(* PLC project Generated.project, CODESYS CODESYS V3.5 SP19 Patch 1 *)
(* stored: creationDateTime 2026-10-27T16:00:37.967713, modificationDateTime 2026-10-27T16:00:37.967713 *)

(* ======================================================================= 📊 ST_Diag_Device — Structure diagnostic d'un esclave ou bus ─────────────────────────────────────────────────────────────── 🎯 Rôle : Structure de donnees d'état, diagnostic et alarme d'un equipement réseau 📄 Doc métier : DOC/AF/AF_Partie-12_Fonction_Diagnostic_v1.4.md ======================================================================= *)
TYPE ST_Diag_Device : STRUCT
  Online : BOOL;  (* Esclave visible sur le bus *)
  Operational : BOOL;  (* Esclave en mode OP (opérationnel) *)
  Error : BOOL;  (* Signal de défaut actif pour cet esclave *)
  ErrorId : WORD;  (* Code défaut détaillé *)
  State : E_Diag_State;  (* Phase courante du cycle de diagnostic *)
  StateAtError : E_Diag_State;  (* Instantané de la phase lors de l'anomalie *)
END_STRUCT;
END_TYPE

(* ======================================================================= 🧩 ST_Fault — Brique socle défaut (2 vues : live + latchée) ─────────────────────────────────────────────────────────────── 🎯 Rôle : porter l'état défaut d'un composant, applicable dans TOUS les cas (acquittable ou non), sans brique warning séparée. • Vue LIVE (Error / ErrorId) : suit la cause, retombe seule à 0. • Vue LATCHÉE (Latched / LatchedId): mémorisée au défaut, reste jusqu'au front Reset. Le choix acquittable / non-acquittable se fait PAR CAUSE (ST_FaultCause.Latching), jamais par bloc. 🔒 Sécurité : interlock TOUJOURS sur la cause brute (Error / ErrorId), jamais sur l'acquittement. Reset TOUJOURS effectif, jamais conditionné (std §9). 🧬 Composition : brique de base réutilisable — sortie de FB, struct métier, GVL. Texte IHM NON stocké ici : dérivé côté IHM depuis LatchedId / ErrorId. 📄 Doc : DOC/STDS/CODE_QUALITY_STANDARDS.md §2quinquies / §9 ======================================================================= *)
TYPE ST_Fault : STRUCT
  Error : BOOL;  (* <-- [DIAG] vue LIVE : au moins une cause présente maintenant *)
  ErrorId : WORD;  (* <-- [DIAG] bitfield des causes présentes maintenant (0 si aucune) *)
  Latched : BOOL;  (* <-- [DIAG] vue LATCHÉE : défaut non acquitté, reste jusqu'au front Reset *)
  LatchedId : WORD;  (* <-- [DIAG] ErrorId figé à l'apparition du défaut, effacé au Reset *)
END_STRUCT;
END_TYPE

(* ======================================================================= 🧩 ST_FaultCause — Cause élémentaire alimentant ST_Fault (socle FB_FaultCore) ─────────────────────────────────────────────────────────────── 🎯 Rôle : une cause exprimée EN CLAIR (BOOL + libellé), sans bitfield ni masque. Le FB métier remplit une liste (ARRAY[0..15] OF ST_FaultCause) ; le socle FB_FaultCore en déduit ST_Fault (vue live + vue latchée). 🔒 Sécurité : interlock TOUJOURS sur Active (cause brute), jamais sur le latch. Latching = TRUE → la cause ARME la vue latchée (défaut à acquitter). Latching = FALSE → la cause n'alimente que la vue live (retombe seule). Fail-safe : une cause laissée à Latching=FALSE reste visible en live — pour la rendre acquittable, il faut le déclarer explicitement. 📄 Doc : DOC/STDS/CODE_QUALITY_STANDARDS.md §2quinquies / §9 ======================================================================= *)
TYPE ST_FaultCause : STRUCT
  Active : BOOL;  (* 1 = cause présente maintenant (interlock sur cette valeur) *)
  Latching : BOOL;  (* 1 = cause à acquitter (arme Latched) ; 0 = live seulement *)
  Texte : STRING;  (* libellé prêt IHM (non stocké dans ST_Fault, dérivé côté IHM) *)
END_STRUCT;
END_TYPE

(* ======================================================================= 🕹️ ST_fbJoystick_AxisCmd — Consigne d'axe normalisée (sortie FB_Joystick) ─────────────────────────────────────────────────────────────── 🎯 Rôle : Structure de consigne d'axe produite par FB_Joystick. 📤 Champs : Enable, StartStop, SpeedTgt (%) + StepTgt (palier 1..5) + direction en bits (DirectionPositive/Negative, AtNeutral). SpeedTgt reste pour l'IHM, StepTgt pour la logique. 📄 Doc métier : DOC/AF/AF_Partie-08_Fonction_Joystick_v2.5.md ======================================================================= *)
TYPE ST_fbJoystick_AxisCmd : STRUCT
  Enable : BOOL;  (* === CONSIGNES DE PILOTAGE AXE === --> [CMD] Autorisation globale pipeline (FALSE=neutralisation, sorties coupees) *)
  StartStop : BOOL;  (* --> [CMD] Validation de mouvement (TRUE=acceleration, FALSE=deceleration/arret) *)
  SpeedTgt : REAL;  (* --> [CMD] Vitesse cible non signee (0...100 %, signe/sens donné par Direction) - IHM *)
  StepTgt : INT;  (* --> [CMD] Palier de vitesse (1..5, 0=arret) - logique/limitations (derive de SpeedTgt) *)
  DirectionNegative : BOOL;  (* --> [CMD] Direction joystick ou intension de gestuelle *)
  DirectionPositive : BOOL;  (* --> [CMD] Direction joystick ou intension de gestuelle *)
  AtNeutral : BOOL;  (* --> [CMD] TRUE si axes en zone morte (position centrale) *)
  Direction : INT;  (* === MONITORING IHM (derive des bits ci-dessus, jamais lu en interlock) === <-- [STAT] Sens -1=Rev / 0=Neutre / +1=Fwd (anim IHM fleche ; lu aussi logique treuils PRG_04) *)
  Deflection : INT;  (* <-- [STAT] Deflexion signee -100..+100 % (anim IHM jauge/barre) *)
END_STRUCT;
END_TYPE

(* ======================================================================= ⚙️ ST_fbJoystick_Cfg — Réglages regroupés de FB_Joystick ─────────────────────────────────────────────────────────────── 🎯 Rôle : porter en un bloc les 5 paramètres de conditionnement du geste (zone morte, temporisations homme-mort, marge défaut capteur). Passé à FB_Joystick via l'entrée `Cfg` — échange bloc IHM / persistant. 🧬 Pattern cfg : aligné sur ST_CycleCfg / ST_WinchCfg (préfixe ST_<Domaine>Cfg, instance persistante dans GVL_PERSISTENT, pont FB_CfgPersistBridge_* à venir). 📄 Doc métier : DOC/AF/AF_Partie-08_Fonction_Joystick_v2.5.md (§5bis) ======================================================================= *)
TYPE ST_fbJoystick_Cfg : STRUCT
  DeadbandRaw : INT := 300;  (* Zone morte en points ADC bruts (0..10000) *)
  NeutralHoldTime : TIME := TIME#100MS;  (* Maintien continu au neutre avant désarmement homme-mort *)
  DeadmanArmHoldTime : TIME := TIME#100MS;  (* Appui continu bouton requis pour armer le geste *)
  DeadmanArmGraceTime : TIME := TIME#3S;  (* Délai de grâce post-armement avant désarmement neutre *)
  RawOutOfRangeMargin : INT := 500;  (* Marge ADC autour des bornes [0..10000] avant défaut capteur (AF08 §5bis) *)
  SpeedStepTable : ST_SpeedStepTable;  (* Les initialiseurs imbriqués de STRUCT (notamment les ARRAY) ne sont pas acceptés par STruCpp/CODESYS dans une déclaration de type. La table est fournie par la configuration persistante de l'appelant. 🪜 Table seuils % -> palier (conversion au joystick, logique FB_Winch §5) *)
  SpeedStepHystMargin : REAL := 2;  (* Marge d'hystérésis palier (%) autour des seuils (anti-oscillation) *)
  Initialized : BOOL := FALSE;  (* 🚦 Flag restauration boot (interne pont FB_CfgPersistBridge_fbJoystick_Cfg) *)
END_STRUCT;
END_TYPE

(* values of E_Diag_State: DISABLED: Désactivé (surveillance non active); READY: Opérationnel réel, pas de défaut; INIT: Initialisation / Recherche de réseau; MONITORING: Surveillance active (états transitoires); ERROR: Anomalie de communication; SIMULATED: Bypass simulation ou bypass réseau IHM — pas le bus réel *)

{attribute 'qualified_only'}
{attribute 'strict'}
TYPE E_Diag_State : (DISABLED := 0, READY := 1, INIT := 2, MONITORING := 3, ERROR := 4, SIMULATED := 5);
END_TYPE

(* ======================================================================= 🪜 ST_SpeedStepTable — Table des paliers de vitesse contacteurs ─────────────────────────────────────────────────────────────── 🎯 Rôle : Structure de configuration des contacteurs et seuils par palier 📄 Doc métier : DOC/AF/AF_Partie-10_Fonction_Winch_v2.1.md ======================================================================= *)
TYPE ST_SpeedStepTable : STRUCT
  P1R1 : BOOL;  (* === PALIER 1 (VITESSE MINIMALE) === Contacteur 1 pour Palier 1 *)
  P1R2 : BOOL;  (* Contacteur 2 pour Palier 1 *)
  P1R3 : BOOL;  (* Contacteur 3 pour Palier 1 *)
  P1R4 : BOOL;  (* Contacteur 4 pour Palier 1 *)
  P2R1 : BOOL;  (* === PALIER 2 === Contacteur 1 pour Palier 2 *)
  P2R2 : BOOL;  (* Contacteur 2 pour Palier 2 *)
  P2R3 : BOOL;  (* Contacteur 3 pour Palier 2 *)
  P2R4 : BOOL;  (* Contacteur 4 pour Palier 2 *)
  P3R1 : BOOL;  (* === PALIER 3 === Contacteur 1 pour Palier 3 *)
  P3R2 : BOOL;  (* Contacteur 2 pour Palier 3 *)
  P3R3 : BOOL;  (* Contacteur 3 pour Palier 3 *)
  P3R4 : BOOL;  (* Contacteur 4 pour Palier 3 *)
  P4R1 : BOOL;  (* === PALIER 4 === Contacteur 1 pour Palier 4 *)
  P4R2 : BOOL;  (* Contacteur 2 pour Palier 4 *)
  P4R3 : BOOL;  (* Contacteur 3 pour Palier 4 *)
  P4R4 : BOOL;  (* Contacteur 4 pour Palier 4 *)
  P5R1 : BOOL;  (* === PALIER 5 (VITESSE MAXIMALE) === Contacteur 1 pour Palier 5 *)
  P5R2 : BOOL;  (* Contacteur 2 pour Palier 5 *)
  P5R3 : BOOL;  (* Contacteur 3 pour Palier 5 *)
  P5R4 : BOOL;  (* Contacteur 4 pour Palier 5 *)
  StepThreshold_Pct : ARRAY[1..5] OF REAL;  (* === SEUILS DE TRANSITION (%) === Seuils de changement de palier (0..100%) *)
END_STRUCT;
END_TYPE

(* ======================================================================= 🕹️ FB_Joystick — Acquisition & conditionnement du geste opérateur ─────────────────────────────────────────────────────────────── 🎯 Rôle : Acquisition 2 axes Hall + bouton homme-mort normatif. Pipeline par axe : FB_AxisScale -> Homme-Mort -> ST_fbJoystick_AxisCmd. 🔒 Sécurité : Armement homme-mort par maintien au neutre. Armement STRICTEMENT conditionné par ArmingPermit (permission externe, vue joystick) ; FALSE = armement bloqué + warning. Désarmement sur neutre prolongé ; le changement de mode / fin de cycle benne est géré par l'externe via ArmingPermit (vue joystick). 📤 Sorties : AxisCmdX/Y (struct = source unique : SpeedTgt NON signee % pour IHM + StepTgt palier 1..5 pour logique + bits sens + Direction -1/0/+1 et Deflection -100..+100 % pour anim IHM), Fault : ST_Fault (socle FB_FaultCore), AtNeutralXY (permis logique), NeutralXAct/YAct (miroirs IHM). 🧬 Contrat : `standard` — pas de struct métier propre → `Fault : ST_Fault` à plat. Pas de `State` (aucune machine d'état), pas de `ST_Lifecycle` (FB synchrone). ⚙️ Réglages regroupés dans `Cfg : ST_fbJoystick_Cfg` (échange bloc IHM / persistant). 📄 Doc métier : DOC/AF/AF_Partie-08_Fonction_Joystick_v2.5.md (F08.01, F08.03-F08.07) ===================================================================== *)
FUNCTION_BLOCK FB_Joystick
  VAR_INPUT
    Enable : BOOL;  (* === CONTRAT STANDARD (Enable + Reset) === --> [CMD] Active la logique du bloc (TRUE=Autorise) *)
    Reset : BOOL;  (* --> [CMD] Acquittement defaut (front, jamais conditionne) *)
    ArmingPermit : BOOL;  (* === PERMIS SECURITE === --> [SAFE] Permission d'armement homme-mort ; FALSE = armement bloqué *)
    DirectInversionPermit : BOOL;  (* --> [SAFE] Inversion Y sans neutre, semi-auto AX8..AX12 et repli du vidage AX15b *)
    BusCanOpenOP : ST_Diag_Device;  (* === ACQUISITION MATERIELLE & DIAGNOSTIC === --> [HW] Etat presence noeud CAN *)
    JoystickOP : ST_Diag_Device;  (* --> [HW] Mode esclave CANopen actif *)
    RawX : INT;  (* --> [HW] Valeur brute axe X (0..10000) *)
    RawY : INT;  (* --> [HW] Valeur brute axe Y (0..10000) *)
    RawButton : BOOL;  (* --> [HW] Etat brut bouton homme-mort *)
    Calibrate : BOOL;  (* === COMMANDES OPERATEUR & CALIBRATION === --> [CMD] Front : lance la calibration (recalage du neutre) *)
    Cfg : ST_fbJoystick_Cfg;  (* === REGLAGES & CONFIGURATION === --> [CFG] Réglages groupés (deadband, temporisations, marge ADC) *)
  END_VAR
  VAR_OUTPUT
    Ready : BOOL;  (* === CONTRAT STANDARD (Ready + Fault) === <-- [STAT] FB pret a fonctionner (Enable + bus OK + pas de defaut late) *)
    Fault : ST_Fault;  (* <-- [DIAG] Brique defaut socle (live + latche), remplie par FB_FaultCore *)
    AxisCmdX : ST_fbJoystick_AxisCmd;  (* === CONSIGNES AXES NORMALISEES === <-- [ACT] Consigne axe X : SpeedTgt (non signee 0..100) + bits sens + Direction/Deflection (monitoring) *)
    AxisCmdY : ST_fbJoystick_AxisCmd;  (* <-- [ACT] Consigne axe Y : SpeedTgt (non signee 0..100) + bits sens + Direction/Deflection (monitoring) *)
    DeadmanArmed : BOOL;  (* === HOMME-MORT === <-- [STAT] Geste arme (bouton maintenu + ArmingPermit) - IHM/diagnostic *)
    ArmingPermitDenied : BOOL;  (* <-- [DIAG] Appui homme-mort refuse (ArmingPermit=FALSE) - warning non latche (F08.08) *)
    AtNeutralXY : BOOL;  (* === ETAT LOGIQUE === <-- [STAT] Les 2 axes en zone morte BRUTE (ScaleX/Y.OutPct=0, AVANT homme-mort) - permis mouvement, LU EN LOGIQUE (PRG_03/04/07) *)
    NeutralXAct : INT;  (* === MIROIRS IHM / TEST === <-- [STAT] Point neutre X calibre courant *)
    NeutralYAct : INT;  (* <-- [STAT] Point neutre Y calibre courant *)
  END_VAR
  VAR_IN_OUT
    NeutralXMem : INT;  (* === RETENTION & CALIBRATION PERSISTANTE === <-> [BUS] Point neutre X persistant global *)
    NeutralYMem : INT;  (* <-> [BUS] Point neutre Y persistant global *)
  END_VAR
  VAR
    CST_DirectionQualificationThreshold_Pct : REAL := 0.1;  (* Seuil % : axe actif (StartStop / bits sens / palier 0) *)
    CST_InversionFlipThreshold_Pct : REAL := 10;  (* Seuil % : sens RETENU pour la détection d'inversion inter-scan. *)
    ScaleX : FB_AxisScale;  (* === SOUS-INSTANCES FB & TIMERS === * [INST] Normalisation et zone morte axe X *)
    ScaleY : FB_AxisScale;  (* * [INST] Normalisation et zone morte axe Y *)
    DeadmanEdge : R_TRIG;  (* * [INST] Detecteur front montant bouton homme-mort *)
    NeutralXYEdge : R_TRIG;  (* * [INST] Front retour simultane X+Y au neutre (libere verrou inversion) *)
    NeutralHoldTimer : TON;  (* * [INST] Temporisation maintien au neutre *)
    DeadmanArmTimer : TON;  (* * [INST] Temporisation maintien bouton armement *)
    DeadmanArmGraceTimer : TON;  (* * [INST] Temporisation delai de grace post-armement *)
    instFault : FB_FaultCore;  (* * [INST] Socle de defaut (liste de causes -> ST_Fault) *)
    SpeedStepHyst1 : HYSTERESIS;  (* * [INST] Decodage % -> palier, seuil 1 (logique FB_Winch §5) *)
    SpeedStepHyst2 : HYSTERESIS;  (* * [INST] Decodage % -> palier, seuil 2 *)
    SpeedStepHyst3 : HYSTERESIS;  (* * [INST] Decodage % -> palier, seuil 3 *)
    SpeedStepHyst4 : HYSTERESIS;  (* * [INST] Decodage % -> palier, seuil 4 *)
    CmdXVal : REAL;  (* === VARIABLES LOCALES INTERNES === . [LOC] Consigne axe X calculee apres filtrage/homme-mort *)
    CmdYVal : REAL;  (* . [LOC] Consigne axe Y calculee apres filtrage/homme-mort *)
    LastCalibrate : BOOL;  (* . [LOC] Memorisation etat precedent commande Calibrate (front) *)
    DeadmanArmPending : BOOL;  (* . [LOC] Armement en cours d'attente de la temporisation maintien *)
    InversionLockActive : BOOL;  (* . [LOC] Verrou retour neutre apres inversion inter-scan directe *)
    PrevDirX : INT;  (* . [LOC] Sens X qualifie au scan precedent (-1, 0, +1) *)
    PrevDirY : INT;  (* . [LOC] Sens Y qualifie au scan precedent (-1, 0, +1) *)
    DirX : INT;  (* . [LOC] Sens X qualifie au scan courant (-1, 0, +1) *)
    DirY : INT;  (* . [LOC] Sens Y qualifie au scan courant (-1, 0, +1) *)
    FlipX : BOOL;  (* . [LOC] Inversion X directe sans echantillon neutre *)
    FlipY : BOOL;  (* . [LOC] Inversion Y directe sans echantillon neutre *)
    RawOutOfRange : BOOL;  (* . [LOC] Surveillance capteur continue (AF08 §5bis) : RawX/RawY hors plage nominale+marge *)
    CalibFail : BOOL;  (* . [LOC] Echec calibration (front Calibrate hors zone) - cause a acquitter (latching) *)
    BusLost : BOOL;  (* . [LOC] Perte liaison bus / device non operationnel - cause live seulement *)
    instCauses : ARRAY[0..15] OF ST_FaultCause;  (* . [LOC] Liste des causes pour le socle FB_FaultCore *)
  END_VAR

            

{region "§1 CAUSES + SOCLE (appele AVANT le gate)"}
// 🎯 CAUSES exprimées en CLAIR (liste ST_FaultCause) — plus de bitfield WORD.
//    - CalibFail : cause A ACQUITTER (Latching=TRUE) -> arme Fault.Latched.
//    - RawOutOfRange / BusLost : cause LIVE seulement (Latching=FALSE) -> Fault.Error, retombe seule.
//    Interlock sur la cause brute ; le socle gère latch/reset.
RawOutOfRange := (RawX < (0 - Cfg.RawOutOfRangeMargin))
              OR (RawX > (10000 + Cfg.RawOutOfRangeMargin))
              OR (RawY < (0 - Cfg.RawOutOfRangeMargin))
              OR (RawY > (10000 + Cfg.RawOutOfRangeMargin));
BusLost := (NOT BusCanOpenOP.Operational OR NOT JoystickOP.Operational);

// Calibration : un front (Calibrate) hors zone -> cause a acquitter. La cause reste active tant que
// les axes sont HORS zone valide [2000..8000] : Reset ne l'efface que si la cause a disparu
// (interlock socle sur la cause brute). Effacee par un Reset avec axes en zone.
IF Calibrate AND NOT LastCalibrate THEN
    IF RawX >= 2000 AND RawX <= 8000 AND RawY >= 2000 AND RawY <= 8000 THEN
        NeutralXMem := RawX;       // memorisation nouvelle position neutre X
        NeutralYMem := RawY;       // memorisation nouvelle position neutre Y
        CalibFail := FALSE;        // calibration valide : plus de cause
    ELSE
        CalibFail := TRUE;         // échec : cause a acquitter (persistante tant que hors zone)
    END_IF;
END_IF;
LastCalibrate := Calibrate;
// Ré-acquisition de la cause (front Reset + cause disparue) : n'efface la cause QUE si les
// axes sont revenus en zone valide. Reste latee tant que hors zone (interlock sur cause brute).
IF Reset AND (RawX >= 2000 AND RawX <= 8000 AND RawY >= 2000 AND RawY <= 8000) THEN
    CalibFail := FALSE;
END_IF;

// Remplissage de la LISTE de causes pour le socle (index 0..2)
// Cause en clair (Active/Latching/Texte) ; 3 causes fixes.
instCauses[0].Active := CalibFail;     instCauses[0].Latching := TRUE;
instCauses[0].Texte := 'Echec calibration joystick (RawX/Y hors zone)';
instCauses[1].Active := RawOutOfRange; instCauses[1].Latching := FALSE;
instCauses[1].Texte := 'Capteur joystick hors plage ADC';
instCauses[2].Active := BusLost;       instCauses[2].Latching := FALSE;
instCauses[2].Texte := 'Perte liaison bus CAN joystick';

// Appel du socle TOUJOURS (meme si le gate RETURN ensuite) : la cause bus doit etre vue.
instFault(Enable := Enable, Reset := Reset, Causes := instCauses);
Fault := instFault.Fault;     // source de verite = socle

// Disponibilite = Enable + bus OK + pas de defaut LATE. Une cause live (bus, capteur) ne latche pas
// -> elle n'entre pas dans Fault.Latched ; le bus est deja couvert par ...OP.Operational ci-dessous.
Ready := Enable AND BusCanOpenOP.Operational AND JoystickOP.Operational AND NOT Fault.Latched;
{endregion}

{region "§2 Gate securite (neutralisation pipeline, n efface pas le statut)"}
// 1. GATE — neutralise le pipeline si indisponible. Le statut a deja ete rempli (zone 0).
IF NOT Enable OR BusLost THEN
    AxisCmdX.Enable := FALSE; AxisCmdX.StartStop := FALSE; AxisCmdX.SpeedTgt := 0.0; AxisCmdX.StepTgt := 0;
    AxisCmdX.DirectionPositive := FALSE; AxisCmdX.DirectionNegative := FALSE; AxisCmdX.AtNeutral := TRUE;
    AxisCmdY.Enable := FALSE; AxisCmdY.StartStop := FALSE; AxisCmdY.SpeedTgt := 0.0; AxisCmdY.StepTgt := 0;
    AxisCmdY.DirectionPositive := FALSE; AxisCmdY.DirectionNegative := FALSE; AxisCmdY.AtNeutral := TRUE;
    AxisCmdX.Direction := 0; AxisCmdX.Deflection := 0;
    AxisCmdY.Direction := 0; AxisCmdY.Deflection := 0;
    AtNeutralXY := TRUE;
    DeadmanArmed := FALSE;
    DeadmanArmPending := FALSE;
    InversionLockActive := FALSE;
    PrevDirX := 0;
    PrevDirY := 0;
    ArmingPermitDenied := FALSE;
    NeutralXYEdge(CLK := FALSE);
    NeutralHoldTimer(IN := FALSE, PT := Cfg.NeutralHoldTime);
    DeadmanArmTimer(IN := FALSE, PT := Cfg.DeadmanArmHoldTime);
    DeadmanArmGraceTimer(IN := FALSE, PT := Cfg.DeadmanArmGraceTime);
    NeutralXAct := NeutralXMem;
    NeutralYAct := NeutralYMem;
    RETURN;
END_IF;
{endregion}

{region "§3 Acquisition + mise a l echelle"}
// Mise a l'echelle (deadband) - le neutre s'evalue sur les 2 axes
ScaleX(RawIn := RawX, Neutral := NeutralXMem, DeadbandRaw := Cfg.DeadbandRaw);
ScaleY(RawIn := RawY, Neutral := NeutralYMem, DeadbandRaw := Cfg.DeadbandRaw);
AtNeutralXY := (ScaleX.OutPct = 0.0) AND (ScaleY.OutPct = 0.0);   // les 2 axes en zone morte - permis mouvement
{endregion}

{region "§4 Armement homme mort"}
// 🔀 Inversion inter-scan : le sens n'est RETENU que si la déflexion dépasse
// CST_InversionFlipThreshold_Pct (>> bruit Hall / bord de deadband). Un aller-retour
// +1<->-1 sans échantillon 0 pose le verrou. Levé exclusivement au front AtNeutralXY.
// RawOutOfRange : lecture capteur non fiable -> aucun sens retenu (le geste est déjà forcé à 0
// par le SEL du pipeline). Une reprise capteur-défaut -> valide ne compte donc pas comme flip.
DirX := 0;
DirY := 0;
IF NOT RawOutOfRange THEN
    IF ScaleX.OutPct > CST_InversionFlipThreshold_Pct THEN
        DirX := 1;
    ELSIF ScaleX.OutPct < -CST_InversionFlipThreshold_Pct THEN
        DirX := -1;
    END_IF;
    IF ScaleY.OutPct > CST_InversionFlipThreshold_Pct THEN
        DirY := 1;
    ELSIF ScaleY.OutPct < -CST_InversionFlipThreshold_Pct THEN
        DirY := -1;
    END_IF;
END_IF;
FlipX := ((PrevDirX = 1) AND (DirX = -1)) OR ((PrevDirX = -1) AND (DirX = 1));
FlipY := ((PrevDirY = 1) AND (DirY = -1)) OR ((PrevDirY = -1) AND (DirY = 1));

NeutralXYEdge(CLK := AtNeutralXY);
IF NeutralXYEdge.Q THEN
    InversionLockActive := FALSE;
END_IF;

IF FlipX OR (FlipY AND NOT (DirectInversionPermit AND DeadmanArmed)) THEN
    InversionLockActive := TRUE;
    DeadmanArmed := FALSE;
    DeadmanArmPending := FALSE;
END_IF;

// Bouton homme-mort : armement par MAINTIEN (Cfg.DeadmanArmHoldTime), independant de la position.
// ⚠️ Un appui PENDANT le verrou d'inversion n'arme PAS de demande : le nouveau front conscient
//    doit survenir APRÈS le retour au neutre (sinon on "pré-charge" le réarmement stick inversé).
DeadmanEdge(CLK := RawButton);
IF DeadmanEdge.Q AND NOT InversionLockActive THEN DeadmanArmPending := TRUE; END_IF;
IF NOT RawButton THEN DeadmanArmPending := FALSE; END_IF;

// Securite : armage UNIQUEMENT si DeadmanArmPending ET ArmingPermit.
DeadmanArmTimer(IN := DeadmanArmPending AND NOT DeadmanArmed AND ArmingPermit AND NOT InversionLockActive, PT := Cfg.DeadmanArmHoldTime);
IF DeadmanArmTimer.Q THEN
    DeadmanArmed := TRUE;
    DeadmanArmPending := FALSE;
END_IF;

// Désarmement externe immédiat : le retrait d'ArmingPermit (changement de mode, fin de cycle
// benne) désarme TOUT DE SUITE le geste — pas d'armement résiduel "surprise" à la ré-acquisition.
IF NOT ArmingPermit THEN
    DeadmanArmed := FALSE;
    DeadmanArmPending := FALSE;
END_IF;

// Avertissement "armage non autorise" (niveau, pendant l'appui non autorise)
ArmingPermitDenied := RawButton AND NOT ArmingPermit;

// Desarmage par maintien au neutre (apres grace)
DeadmanArmGraceTimer(IN := DeadmanArmed, PT := Cfg.DeadmanArmGraceTime);
NeutralHoldTimer(IN := DeadmanArmed AND AtNeutralXY AND DeadmanArmGraceTimer.Q, PT := Cfg.NeutralHoldTime);
IF NeutralHoldTimer.Q THEN DeadmanArmed := FALSE; END_IF;
{endregion}

{region "§5 Pipeline axe X"}
CmdXVal := SEL(DeadmanArmed AND NOT RawOutOfRange, 0.0, ScaleX.OutPct);

AxisCmdX.Enable := NOT RawOutOfRange AND ArmingPermit;
AxisCmdX.SpeedTgt := ABS(CmdXVal);   // NON signee (le sens = bits DirectionPositive/Negative + AxisCmdX.Direction)
AxisCmdX.StartStop := (ABS(CmdXVal) > CST_DirectionQualificationThreshold_Pct);

AxisCmdX.DirectionPositive := (CmdXVal > CST_DirectionQualificationThreshold_Pct);
AxisCmdX.DirectionNegative := (CmdXVal < -CST_DirectionQualificationThreshold_Pct);
AxisCmdX.AtNeutral := NOT AxisCmdX.DirectionPositive AND NOT AxisCmdX.DirectionNegative;
IF AxisCmdX.AtNeutral THEN AxisCmdX.SpeedTgt := 0.0; END_IF;

// Projections monitoring dans le struct (les bits restent la source logique)
IF AxisCmdX.DirectionPositive THEN AxisCmdX.Direction := 1;
ELSIF AxisCmdX.DirectionNegative THEN AxisCmdX.Direction := -1;
ELSE AxisCmdX.Direction := 0; END_IF;
AxisCmdX.Deflection := REAL_TO_INT(CmdXVal);   // deflexion signee -100..+100 % (anim IHM)
{endregion}

{region "§6 Pipeline axe Y et sorties"}
CmdYVal := SEL(DeadmanArmed AND NOT RawOutOfRange, 0.0, ScaleY.OutPct);

AxisCmdY.Enable := NOT RawOutOfRange AND ArmingPermit;
AxisCmdY.SpeedTgt := ABS(CmdYVal);   // NON signee (le sens = bits DirectionPositive/Negative + AxisCmdY.Direction)
AxisCmdY.StartStop := (ABS(CmdYVal) > CST_DirectionQualificationThreshold_Pct);

AxisCmdY.DirectionPositive := (CmdYVal > CST_DirectionQualificationThreshold_Pct);
AxisCmdY.DirectionNegative := (CmdYVal < -CST_DirectionQualificationThreshold_Pct);
AxisCmdY.AtNeutral := NOT AxisCmdY.DirectionPositive AND NOT AxisCmdY.DirectionNegative;
IF AxisCmdY.AtNeutral THEN AxisCmdY.SpeedTgt := 0.0; END_IF;

// 🪜 Decodage consigne % -> palier (logique FB_Winch §5, deplacee au joystick).
//    AxisCmdY.SpeedTgt (%) reste pour l'IHM ; AxisCmdY.StepTgt (1..5, 0=arret) pour la logique/limitations.
SpeedStepHyst1(IN := REAL_TO_INT(AxisCmdY.SpeedTgt), HIGH := REAL_TO_INT(Cfg.SpeedStepTable.StepThreshold_Pct[1] + Cfg.SpeedStepHystMargin), LOW := REAL_TO_INT(Cfg.SpeedStepTable.StepThreshold_Pct[1] - Cfg.SpeedStepHystMargin));
SpeedStepHyst2(IN := REAL_TO_INT(AxisCmdY.SpeedTgt), HIGH := REAL_TO_INT(Cfg.SpeedStepTable.StepThreshold_Pct[2] + Cfg.SpeedStepHystMargin), LOW := REAL_TO_INT(Cfg.SpeedStepTable.StepThreshold_Pct[2] - Cfg.SpeedStepHystMargin));
SpeedStepHyst3(IN := REAL_TO_INT(AxisCmdY.SpeedTgt), HIGH := REAL_TO_INT(Cfg.SpeedStepTable.StepThreshold_Pct[3] + Cfg.SpeedStepHystMargin), LOW := REAL_TO_INT(Cfg.SpeedStepTable.StepThreshold_Pct[3] - Cfg.SpeedStepHystMargin));
SpeedStepHyst4(IN := REAL_TO_INT(AxisCmdY.SpeedTgt), HIGH := REAL_TO_INT(Cfg.SpeedStepTable.StepThreshold_Pct[4] + Cfg.SpeedStepHystMargin), LOW := REAL_TO_INT(Cfg.SpeedStepTable.StepThreshold_Pct[4] - Cfg.SpeedStepHystMargin));

// ⚠️ HYSTERESIS (Util CODESYS) est un hystérésis BAS : OUT=TRUE quand IN<LOW, OUT=FALSE
//    quand IN>HIGH. Pour un décodage ASCENDANT (petite déflexion → palier bas, grande →
//    palier haut) on teste donc `NOT OUT` : palier supérieur seulement une fois IN au-dessus
//    du seuil (bande d'hystérésis LOW..HIGH autour de StepThreshold_Pct[n]).
IF AxisCmdY.SpeedTgt <= CST_DirectionQualificationThreshold_Pct THEN
    AxisCmdY.StepTgt := 0;
ELSE
    AxisCmdY.StepTgt := 1;
    IF NOT SpeedStepHyst1.OUT THEN AxisCmdY.StepTgt := 2; END_IF;
    IF NOT SpeedStepHyst2.OUT THEN AxisCmdY.StepTgt := 3; END_IF;
    IF NOT SpeedStepHyst3.OUT THEN AxisCmdY.StepTgt := 4; END_IF;
    IF NOT SpeedStepHyst4.OUT THEN AxisCmdY.StepTgt := 5; END_IF;
END_IF;

// Projections monitoring dans le struct (les bits restent la source logique)
IF AxisCmdY.DirectionPositive THEN AxisCmdY.Direction := 1;
ELSIF AxisCmdY.DirectionNegative THEN AxisCmdY.Direction := -1;
ELSE AxisCmdY.Direction := 0; END_IF;
AxisCmdY.Deflection := REAL_TO_INT(CmdYVal);   // deflexion signee -100..+100 % (anim IHM)

// Memorisation apres traitement : l'inversion suivante compare deux scans qualifies successifs.
PrevDirX := DirX;
PrevDirY := DirY;

// Miroirs point neutre courant
NeutralXAct := NeutralXMem;
NeutralYAct := NeutralYMem;
{endregion}

          
END_FUNCTION_BLOCK

(* ======================================================================= ⚙️ FB_AxisScale — Normalisation et zone morte d'un axe joystick ─────────────────────────────────────────────────────────────── 🎯 Rôle : Normalise une valeur brute (0..10000) selon le neutre calibré et applique une zone morte en unités brutes (compte ADC). 🛡️ Garde-fou : Saturation stricte de la consigne à +/-100.0 %. 📄 Doc métier : DOC/AF/AF_Partie-08_Fonction_Joystick_v2.5.md (F08.02) ======================================================================= *)
FUNCTION_BLOCK FB_AxisScale
  VAR_INPUT
    RawIn : INT;  (* === ENTRÉES MESURÉES & CONFIGURATION === --> [HW] Valeur brute potentiometre/Hall (0..10000) *)
    Neutral : INT;  (* --> [CFG] Point milieu calibre (compte brut ADC) *)
    DeadbandRaw : INT;  (* --> [CFG] Zone morte en unites brutes ADC (ex: 300) *)
  END_VAR
  VAR_OUTPUT
    OutPct : REAL;  (* === CONSIGNES CALCULÉES === <-- [STAT] Consigne d'axe mise a l'echelle (-100.0..+100.0 %) *)
  END_VAR
  VAR
    Delta : REAL;  (* === VARIABLES LOCALES INTERNES === . [LOC] Amplitude utile de la demi-plage d'axe *)
  END_VAR

            

IF RawIn >= Neutral THEN
    Delta := INT_TO_REAL(10000 - Neutral);
    IF Delta > 0.0 THEN
        OutPct := (INT_TO_REAL(RawIn - Neutral) / Delta) * 100.0;
    ELSE
        OutPct := 0.0;
    END_IF;
ELSE
    Delta := INT_TO_REAL(Neutral);
    IF Delta > 0.0 THEN
        OutPct := (INT_TO_REAL(RawIn - Neutral) / Delta) * 100.0;
    ELSE
        OutPct := 0.0;
    END_IF;
END_IF;

IF ABS(RawIn - Neutral) <= DeadbandRaw THEN
    OutPct := 0.0;
END_IF;

// 🛡️ Limitation de plage : une valeur brute hors plage nominale ne doit jamais
// produire une consigne supérieure à ±100 %. Ce garde-fou protège les
// consommateurs en aval, notamment la translation M3.
OutPct := LIMIT(-100.0, OutPct, 100.0);

          
END_FUNCTION_BLOCK

(* ======================================================================= 🧩 FB_FaultCore — Socle de remplissage de ST_Fault (vue live + vue latchée) ─────────────────────────────────────────────────────────────── 🎯 Rôle : à partir d'une LISTE de causes en clair (ARRAY[0..15] OF ST_FaultCause), produire la brique ST_Fault : • Error / ErrorId : vue LIVE, suit les causes Active, retombe seule. • Latched / LatchedId: vue LATCHÉE, chaque bit figé à l'apparition d'une cause `Active AND Latching`, conservé jusqu'au front Reset. 🔒 Sécurité : - interlock TOUJOURS sur `Causes[i].Active` (cause brute), jamais sur le latch. - Reset TOUJOURS effectif, jamais conditionné (std §9) — agit même Enable=FALSE. - Latching=FALSE → cause visible en LIVE seulement (fail-safe : reste visible). - un défaut laté non acquitté reste publié même FB désactivé (pas d'effacement silencieux sur bascule Enable OFF→ON sans Reset). - une cause à acquitter réapparue re-arme son bit (ré-alarme). 🧬 Un seul socle, réutilisé par tout FB `standard` qui expose un ST_Fault. Pas de State, pas de Warning, pas de texte — hors périmètre de ce socle. 📄 Doc : DOC/STDS/CODE_QUALITY_STANDARDS.md §2quinquies / §9 ======================================================================= *)
FUNCTION_BLOCK FB_FaultCore
  VAR_INPUT
    Enable : BOOL;  (* --> [CMD] Autorisation générale du FB porteur *)
    Reset : BOOL;  (* --> [CMD] Front d'acquittement (jamais conditionné, §9) *)
    Causes : ARRAY[0..15] OF ST_FaultCause;  (* --> [CMD] Liste des causes en clair (Active / Latching / Texte) *)
  END_VAR
  VAR_OUTPUT
    Ready : BOOL;  (* <-- [STAT] FB porteur autorisé (= Enable) *)
    Fault : ST_Fault;  (* <-- [DIAG] Brique défaut (mappée 1:1 sur la sortie du FB porteur) *)
  END_VAR
  VAR
    ResetEdge : R_TRIG;  (* . [LOC] Front montant Reset *)
    Latch : ARRAY[0..15] OF BOOL;  (* . [LOC] Bit laté par cause, jusqu'au Reset *)
    i : INT;  (* . [LOC] Index de parcours de la liste *)
  END_VAR

            

{region "§1 Reset (front, toujours effectif)"}
// Front Reset : efface tous les latches. Jamais conditionné, agit même Enable=FALSE (§9).
Ready := Enable;
ResetEdge(CLK := Reset);
IF ResetEdge.Q THEN
    FOR i := 0 TO 15 DO Latch[i] := FALSE; END_FOR;
END_IF;
{endregion}

{region "§2 Vue LIVE — Error / ErrorId"}
// Bitfield des causes présentes MAINTENANT. Retombe seule à 0 quand les causes disparaissent.
// Non évaluée si Enable=FALSE (pas de lecture de cause hors autorisation).
Fault.ErrorId := 0;
IF Enable THEN
    FOR i := 0 TO 15 DO
        IF Causes[i].Active THEN
            Fault.ErrorId := Fault.ErrorId OR SHL(WORD#1, INT_TO_DWORD(i));
        END_IF;
    END_FOR;
END_IF;
Fault.Error := (Fault.ErrorId <> 0);
{endregion}

{region "§3 Armement des latches (causes à acquitter)"}
// Une cause Active ET Latching arme son bit ; le bit reste jusqu'au front Reset (§1),
// même si la cause disparaît. Réapparition => ré-armement (ré-alarme).
IF Enable THEN
    FOR i := 0 TO 15 DO
        IF Causes[i].Active AND Causes[i].Latching THEN
            Latch[i] := TRUE;
        END_IF;
    END_FOR;
END_IF;
{endregion}

{region "§4 Vue LATCHÉE — Latched / LatchedId"}
// Toujours publiée, y compris Enable=FALSE : un défaut non acquitté reste visible.
Fault.LatchedId := 0;
FOR i := 0 TO 15 DO
    IF Latch[i] THEN
        Fault.LatchedId := Fault.LatchedId OR SHL(WORD#1, INT_TO_DWORD(i));
    END_IF;
END_FOR;
Fault.Latched := (Fault.LatchedId <> 0);
{endregion}

          
END_FUNCTION_BLOCK
